KUKA KRL data list: LAB_PATHS.dat

&ACCESS RVP
&REL 1
DEFDAT LAB_PATHS PUBLIC
  DECL E6AXIS A_HOME={A1 0,A2 -90,A3 90,A4 0,A5 0,A6 0,E1 0,E2 0,E3 0,E4 0,E5 0,E6 0}
  DECL E6POS P_START={X 1900,Y -200,Z 1200,A 180,B 0,C 180,S 2,T 2,E1 0,E2 0,E3 0,E4 0,E5 0,E6 0}
  DECL E6POS P_AUX={X 1950,Y -100,Z 1200,A 180,B 0,C 180,S 2,T 2,E1 0,E2 0,E3 0,E4 0,E5 0,E6 0}
  DECL E6POS P_ARC_END={X 1900,Y 0,Z 1200,A 180,B 0,C 180,S 2,T 2,E1 0,E2 0,E3 0,E4 0,E5 0,E6 0}
  DECL E6POS P_SPLINE_1={X 1900,Y 100,Z 1200,A 180,B 0,C 180,S 2,T 2,E1 0,E2 0,E3 0,E4 0,E5 0,E6 0}
  DECL E6POS P_SPLINE_2={X 1950,Y 150,Z 1200,A 180,B 0,C 180,S 2,T 2,E1 0,E2 0,E3 0,E4 0,E5 0,E6 0}
  DECL E6POS P_SPLINE_AUX={X 1950,Y 200,Z 1200,A 180,B 0,C 180,S 2,T 2,E1 0,E2 0,E3 0,E4 0,E5 0,E6 0}
  DECL E6POS P_SPLINE_END={X 1900,Y 250,Z 1200,A 180,B 0,C 180,S 2,T 2,E1 0,E2 0,E3 0,E4 0,E5 0,E6 0}
ENDDAT
